FUNCTION_BLOCK "Keller_pressure_transmitters"
{ S7_Optimized_Access := 'TRUE' }
VERSION : 0.1
   VAR_INPUT
      unit : USInt;
   END_VAR

   VAR_IN_OUT
      mb : "udt_mb";
   END_VAR

   VAR
      common : "udt_mb_common";
      data : Struct
         pressure_sensor_1 : Real;
         pressure_sensor_2 : Real;
         temperature : Real;
         temperature_sensor_1 : Real;
         temperature_sensor_2 : Real;
      END_STRUCT;
   END_VAR


BEGIN
	// Keller, Series 30 and Series 40 - pressure transmitters

	// Warning: Block is NOT tested !

	// Doc:
	// http://www.keller-druck.com/picts/pdf/engl/comm_protocol_e.pdf

	"mb_device_header"(common := #common, mb := #mb);

	"mb_query"(unit := #unit,
	           fc := #mb.c.read.holding_reg,
	           d_addr := 2,
	           d_len := #mb.c.auto_len,
	           data := #data,
	           mb := #mb);

	"mb_device_footer"(common := #common, mb := #mb);

	IF #common.out.communication_error THEN
	    #data.pressure_sensor_1 := 0;
	    #data.pressure_sensor_2 := 0;
	    #data.temperature := 0;
	    #data.temperature_sensor_1 := 0;
	    #data.temperature_sensor_2 := 0;
	END_IF;

END_FUNCTION_BLOCK

